// TIA Portal project "SCADA_FINAL" (V16)

(* hardware
DEVICE "S71500/ET200MP station_1"  S7-1500 station
   slot 0: "Rail_0"  Rack  6ES7 590-1***0-0AA0
   slot 1: "PLC_1"  CPU 1511-1 PN  6ES7 511-1AK02-0AB0  V2.8
      slot 3: "CPU display_1"  6ES7591-1AA00-0AA0
      slot 32768: "PROFINET interface_1"  X1
         slot 32769: "Port_1"  X1 P1
         slot 32770: "Port_2"  X1 P2
      slot 34817: "Virtual CP interface port_1"  Virtual CP interface port  Virtual CP interface port
DEVICE "PC-System_1"  SIMATIC PC station
   slot 0: "SIMATIC PC station"  Rail  SIMATIC PC-Station  V1.0
      slot 125: "Stationmanager"  Station_Manager  V6.0.4
   slot 1: "HMI_RT_1"  WinCC RT Professional  6AV2 105-0xxxx-xxxx  16.0.0.0
   slot 2: "IE general_1"  IE General  IE_CP  V8.2.0
*)

// ===== PLC "PLC_1"  CPU 1511-1 PN =====

VAR_GLOBAL   // PLC tag table "Default tag table"
   "Clock_Byte" AT %MB0 : Byte;
   "Clock_10Hz" AT %M0.0 : Bool;
   "Clock_5Hz" AT %M0.1 : Bool;
   "Clock_2.5Hz" AT %M0.2 : Bool;
   "Clock_2Hz" AT %M0.3 : Bool;
   "Clock_1.25Hz" AT %M0.4 : Bool;
   "Clock_1Hz" AT %M0.5 : Bool;
   "Clock_0.625Hz" AT %M0.6 : Bool;
   "Clock_0.5Hz" AT %M0.7 : Bool;
   "LEVEL" AT %MW100 : Int;
   "LEVEL1" AT %MW102 : Int;
   "System_Byte" AT %MB1 : Byte;
   "FirstScan" AT %M1.0 : Bool;
   "DiagStatusUpdate" AT %M1.1 : Bool;
   "AlwaysTRUE" AT %M1.2 : Bool;
   "AlwaysFALSE" AT %M1.3 : Bool;
END_VAR

DATA_BLOCK "M_1_1"   // DB1
{ S7_Optimized_Access := 'FALSE' }
VERSION : 0.1
// stored: InstanceOfName MOTOR
"MOTOR"
BEGIN
END_DATA_BLOCK

DATA_BLOCK "M_1_2"   // DB2
{ S7_Optimized_Access := 'FALSE' }
VERSION : 0.1
// stored: InstanceOfName MOTOR
"MOTOR"
BEGIN
END_DATA_BLOCK

DATA_BLOCK "M_2_1"   // DB3
{ S7_Optimized_Access := 'FALSE' }
VERSION : 0.1
// stored: InstanceOfName MOTOR
"MOTOR"
BEGIN
END_DATA_BLOCK

DATA_BLOCK "M_2_2"   // DB4
{ S7_Optimized_Access := 'FALSE' }
VERSION : 0.1
// stored: InstanceOfName MOTOR
"MOTOR"
BEGIN
END_DATA_BLOCK

DATA_BLOCK "MIXER"   // DB5
{ S7_Optimized_Access := 'FALSE' }
VERSION : 0.1
// stored: InstanceOfName MOTOR
"MOTOR"
BEGIN
END_DATA_BLOCK

DATA_BLOCK "V_3_1"   // DB6
{ S7_Optimized_Access := 'FALSE' }
VERSION : 0.1
// stored: InstanceOfName MOTOR
"MOTOR"
BEGIN
END_DATA_BLOCK

DATA_BLOCK "V_3_2"   // DB7
{ S7_Optimized_Access := 'FALSE' }
VERSION : 0.1
// stored: InstanceOfName MOTOR
"MOTOR"
BEGIN
END_DATA_BLOCK

DATA_BLOCK "CONTROL_PANEL"   // DB9
{ S7_Optimized_Access := 'FALSE' }
VERSION : 0.1
   VAR
      HI1 : Bool;
      LO1 : Bool;
      HI : Bool;
      LO : Bool;
      START : Bool;
      STOP : Bool;
   END_VAR
BEGIN
END_DATA_BLOCK

DATA_BLOCK "Auto1"   // DB10
{ S7_Optimized_Access := 'FALSE' }
VERSION : 0.1
   VAR
      START : Bool;
      STOP : Bool;
      HI1 : Bool;
      LO1 : Bool;
      M_1_1 : Bool;
      M_1_2 : Bool;
      S0 : Bool;
      S1 : Bool;
      S2 : Bool;
      S3 : Bool;
      T00 : Bool;
      T01 : Bool;
      T12 : Bool;
      T10 : Bool;
      T20 : Bool;
      T23 : Bool;
      T31 : Bool;
      T30 : Bool;
   END_VAR
BEGIN
END_DATA_BLOCK

DATA_BLOCK "Auto2"   // DB11
{ S7_Optimized_Access := 'FALSE' }
VERSION : 0.1
   VAR
      HI : Bool;
      LO : Bool;
      M_2 : Bool;
      V_3 : Bool;
      MIXER : Bool;
      S0 : Bool;
      S1 : Bool;
      S2 : Bool;
      S3 : Bool;
      S4 : Bool;
      T00 : Bool;
      T01 : Bool;
      T10 : Bool;
      T14 : Bool;
      T12 : Bool;
      T23 : Bool;
      T20 : Bool;
      T30 : Bool;
      T31 : Bool;
      T41 : Bool;
   END_VAR
BEGIN
END_DATA_BLOCK

DATA_BLOCK "DisplayScreen"   // DB14
{ S7_Optimized_Access := 'FALSE' }
VERSION : 0.1
   VAR
      Level : Int;
      Level1 : Int;
   END_VAR
BEGIN
END_DATA_BLOCK

// folder: System blocks/Program resources

DATA_BLOCK "T10S"   // DB12
{ S7_Optimized_Access := 'TRUE' }
AUTHOR : Simatic
FAMILY : IEC
NAME : IEC_TMR
VERSION : 1.0
// stored: InstanceOfName IEC_TIMER
"IEC_TIMER"
BEGIN
END_DATA_BLOCK

DATA_BLOCK "T10S1"   // DB13
{ S7_Optimized_Access := 'TRUE' }
AUTHOR : Simatic
FAMILY : IEC
NAME : IEC_TMR
VERSION : 1.0
// stored: InstanceOfName IEC_TIMER
"IEC_TIMER"
BEGIN
END_DATA_BLOCK

// folder: (top level)

FUNCTION_BLOCK "MOTOR"   // FB1, SCL
{ S7_Optimized_Access := 'FALSE' }
VERSION : 0.1
   VAR_INPUT
      MODE : Int;
      START : Bool;
      STOP : Bool;
      RUNCONDITION : Bool;
      STOPCONDITION : Bool;
      RUNFEEDBACK : Bool;
      RESET : Bool;
   END_VAR
   VAR_OUTPUT
      CMD : Bool;
      FAULT : Bool;
   END_VAR
   VAR
      DELAY_CMD : TON_TIME;
   END_VAR
BEGIN
   IF #MODE = 1 THEN
       // Statement section IF
       #CMD := (#START OR #CMD) AND NOT #STOP AND NOT #FAULT;
   END_IF;
   IF #MODE = 2 THEN
       // Statement section IF
       #CMD := (#RUNCONDITION OR #CMD)AND NOT #STOPCONDITION AND NOT #FAULT;
   END_IF;

   #DELAY_CMD(IN:=#CMD,
              PT:=T#5S);
   IF #DELAY_CMD.Q AND NOT #RUNFEEDBACK THEN
       // Statement section IF
       #FAULT := 1;
   END_IF;

   IF #RESET THEN
       // Statement section IF
       #FAULT := 0;
   END_IF;
END_FUNCTION_BLOCK

ORGANIZATION_BLOCK "Main"   // OB1, FBD, ProgramCycle
TITLE = "Main Program Sweep (Cycle)"
{ S7_Optimized_Access := 'TRUE' }
VERSION : 0.1
   VAR_INPUT
      Initial_Call : Bool;   // Initial call of this OB
      Remanence : Bool;   // =True, if remanent data are available
   END_VAR
BEGIN

REGION Network 1
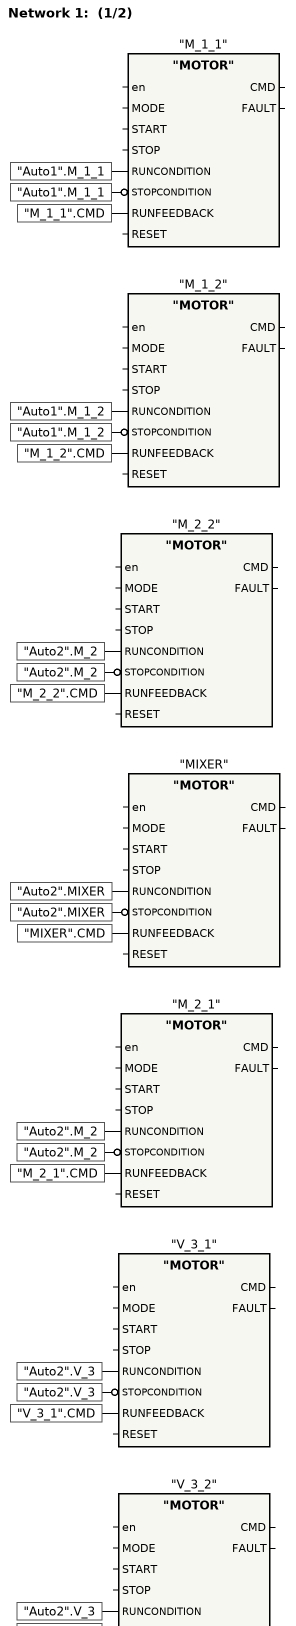
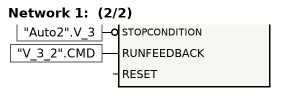
   "M_1_1"(RUNCONDITION := "Auto1".M_1_1, STOPCONDITION := NOT "Auto1".M_1_1, RUNFEEDBACK := "M_1_1".CMD);   // "MOTOR"
   "M_1_2"(RUNCONDITION := "Auto1".M_1_2, STOPCONDITION := NOT "Auto1".M_1_2, RUNFEEDBACK := "M_1_2".CMD);   // "MOTOR"
   "M_2_2"(RUNCONDITION := "Auto2".M_2, STOPCONDITION := NOT "Auto2".M_2, RUNFEEDBACK := "M_2_2".CMD);   // "MOTOR"
   "MIXER"(RUNCONDITION := "Auto2".MIXER, STOPCONDITION := NOT "Auto2".MIXER, RUNFEEDBACK := "MIXER".CMD);   // "MOTOR"
   "M_2_1"(RUNCONDITION := "Auto2".M_2, STOPCONDITION := NOT "Auto2".M_2, RUNFEEDBACK := "M_2_1".CMD);   // "MOTOR"
   "V_3_1"(RUNCONDITION := "Auto2".V_3, STOPCONDITION := NOT "Auto2".V_3, RUNFEEDBACK := "V_3_1".CMD);   // "MOTOR"
   "V_3_2"(RUNCONDITION := "Auto2".V_3, STOPCONDITION := NOT "Auto2".V_3, RUNFEEDBACK := "V_3_2".CMD);   // "MOTOR"
END_REGION
END_ORGANIZATION_BLOCK

ORGANIZATION_BLOCK "SIM"   // OB123, SCL, ProgramCycle
TITLE = "Main Program Sweep (Cycle)"
{ S7_Optimized_Access := 'TRUE' }
VERSION : 0.1
   VAR_INPUT
      Initial_Call : Bool;   // Initial call of this OB
      Remanence : Bool;   // =True, if remanent data are available
   END_VAR
BEGIN
   "R_TRIG_DB"(CLK:="Clock_1Hz");

   IF "M_1_1".RUNFEEDBACK AND "R_TRIG_DB".Q THEN
       // Statement section IF
       "LEVEL1" := "LEVEL1" + 1;
       IF "LEVEL1" >= 100 THEN
           // Statement section IF
           "LEVEL1" := 100;
       END_IF;
   END_IF;

   IF "M_1_2".RUNFEEDBACK AND "R_TRIG_DB".Q THEN
       // Statement section IF
       "LEVEL1" := "LEVEL1" + 1;
       IF "LEVEL1" >= 100 THEN
           // Statement section IF
           "LEVEL1" := 100;
       END_IF;
   END_IF;

   IF "M_2_1".RUNFEEDBACK AND "R_TRIG_DB".Q THEN
       // Statement section IF
       "LEVEL" := "LEVEL" + 1;
       "LEVEL1" := "LEVEL1" - 1;
       IF "LEVEL" >= 100 THEN
           // Statement section IF
           "LEVEL" := 100;
       END_IF;
       IF "LEVEL1" <=0 THEN
           // Statement section IF
           "LEVEL1" := 0;
       END_IF;

   END_IF;

   IF "M_2_2".RUNFEEDBACK AND "R_TRIG_DB".Q THEN
       // Statement section IF
       "LEVEL" := "LEVEL" + 1;
       IF "LEVEL" >= 100 THEN
           // Statement section IF
           "LEVEL" := 100;
       END_IF;
   END_IF;

   IF "V_3_1".RUNFEEDBACK AND "R_TRIG_DB".Q THEN
       // Statement section IF
       "LEVEL" := "LEVEL" - 1;
       IF "LEVEL" <= 0 THEN
           // Statement section IF
           "LEVEL" := 0;
       END_IF;
   END_IF;

   IF "V_3_2".RUNFEEDBACK AND "R_TRIG_DB".Q THEN
       // Statement section IF
       "LEVEL" := "LEVEL" - 1;
       IF "LEVEL" <= 0 THEN
           // Statement section IF
           "LEVEL" := 0;
       END_IF;
   END_IF;

   IF "LEVEL" >= 99 THEN
       // Statement section IF
       "CONTROL_PANEL".HI := TRUE;
   ELSE
       "CONTROL_PANEL".HI := FALSE;
   END_IF;

   IF "LEVEL1" >= 99 THEN
       // Statement section IF
       "CONTROL_PANEL".HI1 := TRUE;
   ELSE
       "CONTROL_PANEL".HI1 := FALSE;
   END_IF;

   IF "LEVEL" <= 1 THEN
       // Statement section IF
       "CONTROL_PANEL".LO := TRUE;
   ELSE
       "CONTROL_PANEL".LO := FALSE;
   END_IF;

   IF "LEVEL1" <= 1 THEN
       // Statement section IF
       "CONTROL_PANEL".LO1 := TRUE;
   ELSE
       "CONTROL_PANEL".LO1 := FALSE;
   END_IF;

   IF "LEVEL1" < 5 THEN
       // Statement section IF
       "M_2_1".CMD:= FALSE;
       "M_2_2".CMD := FALSE;
   END_IF;


   "DisplayScreen".Level := "LEVEL";
   "DisplayScreen".Level1 := "LEVEL1";
END_ORGANIZATION_BLOCK

ORGANIZATION_BLOCK "AutoMode"   // OB124, SCL, ProgramCycle
TITLE = "Main Program Sweep (Cycle)"
{ S7_Optimized_Access := 'TRUE' }
VERSION : 0.1
   VAR_INPUT
      Initial_Call : Bool;   // Initial call of this OB
      Remanence : Bool;   // =True, if remanent data are available
   END_VAR
BEGIN
   "T10S".TON(IN:="Auto1".S1,
              PT:=T#10s);
   "T10S1".TON(IN:="Auto2".S2,
               PT:=T#10s);
   //transition logics
   "Auto1".T00 := "FirstScan";
   "Auto1".T01 := "Auto1".S0 AND "CONTROL_PANEL".START;
   "Auto1".T10 := "Auto1".S1 AND "CONTROL_PANEL".STOP;
   "Auto1".T12 := "Auto1".S1 AND "T10S".Q;
   "Auto1".T20 := "Auto1".S2 AND "CONTROL_PANEL".STOP;
   "Auto1".T23 := "Auto1".S2 AND "CONTROL_PANEL".HI1;
   "Auto1".T30 := "Auto1".S3 AND "CONTROL_PANEL".STOP;
   "Auto1".T31 := "Auto1".S3 AND "CONTROL_PANEL".LO1;

   //state logics
   "Auto1".S0 := ("Auto1".S0 OR "Auto1".T00 OR "Auto1".T10 OR "Auto1".T20 OR "Auto1".T30) AND NOT "Auto1".T01;
   "Auto1".S1 := ("Auto1".S1 OR "Auto1".T01 OR "Auto1".T31) AND NOT "Auto1".T10 AND NOT "Auto1".T12;
   "Auto1".S2 := ("Auto1".S2 OR "Auto1".T12) AND NOT "Auto1".T20 AND NOT "Auto1".T23;
   "Auto1".S3 := ("Auto1".S3 OR "Auto1".T23) AND NOT "Auto1".T30 AND NOT "Auto1".T31;

   //output logic 
   "Auto1".M_1_1 := "Auto1".S1 OR "Auto1".S2;
   "Auto1".M_1_2 := "Auto1".S2;


   //transition logic
   "Auto2".T00 := "FirstScan";
   "Auto2".T01 := "Auto2".S0 AND "CONTROL_PANEL".START;
   "Auto2".T10 := "Auto2".S1 AND "CONTROL_PANEL".STOP;
   "Auto2".T12 := "Auto2".S1 AND "CONTROL_PANEL".HI;
   "Auto2".T14 := "Auto2".S1 AND "CONTROL_PANEL".LO1;
   "Auto2".T20 := "Auto2".S2 AND "CONTROL_PANEL".STOP;
   "Auto2".T23 := "Auto2".S2 AND "T10S1".Q;
   "Auto2".T30 := "Auto2".S3 AND "CONTROL_PANEL".STOP;
   "Auto2".T31 := "Auto2".S3 AND "CONTROL_PANEL".LO;
   "Auto2".T41 := "Auto2".S4 AND "CONTROL_PANEL".LO1;
   //State logics
   "Auto2".S0 := ("Auto2".S0 OR "Auto2".T00 OR "Auto2".T10 OR "Auto2".T20 OR "Auto2".T30) AND NOT "Auto2".T01;
   "Auto2".S1 := ("Auto2".S1 OR "Auto2".T01 OR "Auto2".T31 OR "Auto2".T41) AND NOT "Auto2".T10 AND NOT "Auto2".T12 AND NOT "Auto2".T14;
   "Auto2".S2 := ("Auto2".S2 OR "Auto2".T12) AND NOT "Auto2".T23 AND NOT "Auto2".T20;
   "Auto2".S3 := ("Auto2".S3 OR "Auto2".T23) AND NOT "Auto2".T30 AND NOT "Auto2".T31;
   "Auto2".S4 := ("Auto2".S4 OR "Auto2".T14) AND NOT "Auto2".T41;
   //output logics
   "Auto2".M_2 := "Auto2".S1;
   "Auto2".MIXER := "Auto2".S2;
   "Auto2".V_3 := "Auto2".S3;
END_ORGANIZATION_BLOCK